TYPE E_PrintSelection :
(
	// Binary Enum. Print A&B = PrintHeadA | PrintHeadB = 0x03
	None		 	:= 16#00,
	PrintHeadA		:= 16#01,
	PrintHeadB		:= 16#02,
	MAX_E_PrintSelection
);
END_TYPE

(* stored: Version 1.1.0.1, ProductVersion 3.1.0.24
   DUT E_PrintSelection: Id {d1efabbd-b801-4ea2-b5f0-2dd1b77b67ff} *)
